**Example:**
```
iterator.reset();
WHILE(iterator.moveNext())DO
	foo := iterator.current.hashCode;
	bar := iterator.current.name;
END_WHILE
```

.. <legal notes>

legal notes
=================
| SPDX-FileCopyrightText: © 2022 ekvip automation GmbH <info@ekvip.de>
| SPDX-License-Identifier: Apache-2.0
| For details check: Apache-2.0_

.. _Apache-2.0: https://www.apache.org/licenses/LICENSE-2.0

.. </legal notes>

*)
METHOD reset
VAR CONSTANT
	NULL :__XWORD := 0;
END_VAR
THIS^.iterate(execute := FALSE);
THIS^.nextIndex := 0;
THIS^.currentObject := NULL;
END_METHOD

END_FUNCTION_BLOCK

// ---- Utils/FastSwap.TcPOU
(*
## Short summary

Fast element swap operation of two given pointers, optimized for performance.

.. <legal notes>

legal notes
=================
| SPDX-FileCopyrightText: © 2025 ekvip automation GmbH <info@ekvip.de>
| SPDX-License-Identifier: Apache-2.0
| For details check: Apache-2.0_

.. _Apache-2.0: https://www.apache.org/licenses/LICENSE-2.0

.. </legal notes>



*)

FUNCTION FastSwap
VAR_INPUT
	object1 :POINTER TO __XWORD;
	object2 :POINTER TO __XWORD;
END_VAR

RETURN(object1 = object2);
RETURN(object1 = 0 OR object2 = 0);
object1^ := object2^ XOR object1^;
object2^ := object2^ XOR object1^;
object1^ := object2^ XOR object1^;

END_FUNCTION

// ---- Lists/ArrayList/ArrayListResizingStrategy/CubicRootResizing.TcPOU
(*

## Short summary

This resizing strategy increases an capacity by a geometric factor of the cubic root of 2 (~1.26).
After three consecutive growth steps, the capacity approximately doubles, which improves the chance of reusing previously freed memory blocks and helps to reduce heap fragmentation.
The strategy is well-suited for memory-constrained or embedded environments where efficient memory reuse is more important than minimizing the number of reallocation operations.
For downsizing the capacity is reduced if the new size is less then 25 % of the current capacity. 

.. <legal notes>

legal notes
=================
| SPDX-FileCopyrightText: © 2025 ekvip automation GmbH <info@ekvip.de>
| SPDX-License-Identifier: Apache-2.0
| For details check: Apache-2.0_

.. _Apache-2.0: https://www.apache.org/licenses/LICENSE-2.0

.. </legal notes>

*)

{attribute 'enable_dynamic_creation'}
FUNCTION_BLOCK CubicRootResizing EXTENDS CNM_AbstractObject.Object IMPLEMENTS CNM_CollectionInterfaces.IResizingStrategy
VAR CONSTANT
	(* cubic root of 2 *)
	GROW_FACTOR :REAL := 1.259921049894873165;
END_VAR

(*

## Short summary

This abstract property returns the class name of the concrete object, 
which is useful for logging/debugging purpose.

.. <legal notes>

legal notes
=================
| SPDX-FileCopyrightText: © 2022 ekvip automation GmbH <info@ekvip.de>
| SPDX-License-Identifier: Apache-2.0
| For details check: Apache-2.0_

.. _Apache-2.0: https://www.apache.org/licenses/LICENSE-2.0

.. </legal notes>

*)
PROPERTY className : CNM_AbstractObject.ClassName
GET
className := 'CNM_Collections.CubicRootResizing';
END_GET
END_PROPERTY

(*

## Short summary

The method takes the requested size and the current capacity as input and determines the next suitable capacity value based on the implemented resizing strategy.
The resulting capacity is returned as newCapacity.
It returns true when a downsizing is needed within the used strategy, false if no resizing is needed.

.. <legal notes>

legal notes
=================
| SPDX-FileCopyrightText: © 2025 ekvip automation GmbH <info@ekvip.de>
| SPDX-License-Identifier: Apache-2.0
| For details check: Apache-2.0_

.. _Apache-2.0: https://www.apache.org/licenses/LICENSE-2.0

.. </legal notes>



*)
METHOD getDownscaledCapacity : BOOL
VAR_INPUT
	(* the new size that is needed *)
	requestedSize	: UDINT;
	(* the current actual size of the container *)
	currentCapacity	: UDINT;
END_VAR
VAR_OUTPUT
	(* the calculated size of the container *)
	newCapacity	: UDINT;
END_VAR
VAR CONSTANT
	SHRINKING_THRESHOLD_MULTIPLIER :UDINT := 3;
END_VAR
IF (requestedSize < THIS^.initialSize) OR_ELSE (currentCapacity = 0) THEN 
	newCapacity := THIS^.initialSize; 
ELSE 
	newCapacity := currentCapacity;  
	// gradual shrink by cubic root of 0.5 with threshold 
	WHILE ( newCapacity > SHRINKING_THRESHOLD_MULTIPLIER*requestedSize ) DO
		newCapacity := TO_UDINT(TO_REAL(newCapacity) / THIS^.GROW_FACTOR);
	END_WHILE
END_IF;

getDownscaledCapacity := (newCapacity <> currentCapacity);
END_METHOD

(*

## Short summary

The method takes the requested size and the current capacity as input and determines the next suitable capacity value based on the implemented resizing strategy.
The resulting capacity is returned as newCapacity. 
It returns true when a resizing is needed wihtin the used strategy, false if no resizing is needed.

.. <legal notes>

legal notes
=================
| SPDX-FileCopyrightText: © 2025 ekvip automation GmbH <info@ekvip.de>
| SPDX-License-Identifier: Apache-2.0
| For details check: Apache-2.0_

.. _Apache-2.0: https://www.apache.org/licenses/LICENSE-2.0

.. </legal notes>



*)
METHOD getUpscaledCapacity : BOOL
VAR_INPUT
	(* the new size that is needed *)
	requestedSize	: UDINT;
	(* the current actual size of the container *)
	currentCapacity	: UDINT;
END_VAR
VAR_OUTPUT
	(* the calculated size of the container *)
	newCapacity	: UDINT;
END_VAR
IF (requestedSize < THIS^.initialSize) THEN
	newCapacity := THIS^.initialSize;
ELSE
	newCapacity := SEL((currentCapacity = 0), newCapacity := currentCapacity, newCapacity := THIS^.initialSize);
	WHILE (newCapacity < requestedSize) DO
		newCapacity := TO_UDINT(TO_REAL(newCapacity) * THIS^.GROW_FACTOR);
	END_WHILE
END_IF
getUpscaledCapacity := (newCapacity <> currentCapacity);
END_METHOD

(*

## Short summary

This property returns an inital size for an empty new array. 

.. <legal notes>

legal notes
=================
| SPDX-FileCopyrightText: © 2025 ekvip automation GmbH <info@ekvip.de>
| SPDX-License-Identifier: Apache-2.0
| For details check: Apache-2.0_

.. _Apache-2.0: https://www.apache.org/licenses/LICENSE-2.0

.. </legal notes>



*)

PROPERTY initialSize : UDINT
GET
initialSize := 8;
END_GET
END_PROPERTY

END_FUNCTION_BLOCK

// ---- Appliers/classes/ChainedApplier.TcPOU
(*

## Short summary

An abstract class to implement the logic of Appliers for forEach. Users only need to implement apply in inherited class and should not change any other method.

.. <legal notes>

legal notes
=================
| SPDX-FileCopyrightText: © 2022 ekvip automation GmbH <info@ekvip.de>
| SPDX-License-Identifier: Apache-2.0
| For details check: Apache-2.0_

.. _Apache-2.0: https://www.apache.org/licenses/LICENSE-2.0

.. </legal notes>



*)

{attribute 'enable_dynamic_creation'}
FUNCTION_BLOCK FINAL ChainedApplier EXTENDS AbstractDisposableContainer IMPLEMENTS CNM_CollectionInterfaces.IChainedApplier
VAR
	object :CNM_AbstractObject.IObject;
END_VAR
VAR
	myactions			:ApplierList();
END_VAR

(*

## Short summary

Method to accept an object.
**Example:**
```
NumberIncrementer.accept(Number);
```

.. <legal notes>

legal notes
=================
| SPDX-FileCopyrightText: © 2022 ekvip automation GmbH <info@ekvip.de>
| SPDX-License-Identifier: Apache-2.0
| For details check: Apache-2.0_

.. _Apache-2.0: https://www.apache.org/licenses/LICENSE-2.0

.. </legal notes>



*)
METHOD accept : CNM_ReturnTypes.SingleExecutionResult
VAR_INPUT
	(*object to accept*)
	object	: CNM_AbstractObject.IObject;
END_VAR
IF(THIS^.isObjectValid(object))THEN
	THIS^.object := object;
	accept := CNM_ReturnTypes.SingleExecutionResult.SUCCESS;
ELSE
	accept := CNM_ReturnTypes.SingleExecutionResult.ERROR;	
END_IF
END_METHOD

(*

## Short summary

This property returns a list of actions/operations performed by this applier.

.. <legal notes>

legal notes
=================
| SPDX-FileCopyrightText: © 2022 ekvip automation GmbH <info@ekvip.de>
| SPDX-License-Identifier: Apache-2.0
| For details check: Apache-2.0_

.. _Apache-2.0: https://www.apache.org/licenses/LICENSE-2.0

.. </legal notes>

*)

PROPERTY actions :CNM_CollectionInterfaces.IApplierList
GET
actions := THIS^.myactions;
END_GET
END_PROPERTY

(*

## Short summary

Method to concat actions perfomed on an object. This way two (or more) Actions can be performed on data with one foreach.
All concatinated appliers can be cleared with THIS^.clear();
**Example:**
You want to double your numbers and then increment them, you would write:
```
ConcreteDoubleApplier.andThen(ConcreteIncrementApplier);
```
If you have a list with 1 2 3, after a forEach with this Applier the list will be transformed to: 3 5 7.

**Warning:**
    It is possible to create infinite loops using andThen. For example: A1.andThen(A2).andThen(A1)
	The program will go into unknown behaviour if this occurs and the foreach call may or may not work as you intended.

.. <legal notes>

legal notes
=================
| SPDX-FileCopyrightText: © 2022 ekvip automation GmbH <info@ekvip.de>
| SPDX-License-Identifier: Apache-2.0
| For details check: Apache-2.0_

.. _Apache-2.0: https://www.apache.org/licenses/LICENSE-2.0

.. </legal notes>


**Return:** ``THIS^`` `IApplier`

*)

METHOD FINAL andThen :CNM_CollectionInterfaces.IChainedApplier
VAR_INPUT
	(*the applier to be used on each object*)
	applier			:CNM_CollectionInterfaces.IApplier;
END_VAR
VAR
	chained 		:CNM_CollectionInterfaces.IChainedApplier;
	clonedActions	:CNM_CollectionInterfaces.ICollection;
	cloneObj 		:CNM_AbstractObject.IObject;
	pList 			:POINTER TO ApplierList;
END_VAR
IF(THIS^.isObjectValid(applier) AND_THEN THIS^.isObjectValid(THIS^.myactions))THEN
	IF __QUERYINTERFACE(applier, chained) THEN
		IF (chained.actions.count > 1) THEN
			IF(NOT THIS^.isEqual(applier))THEN
				__QUERYPOINTER(chained.actions, pList);
				THIS^.myactions.addAppliers(pList^.list);
			ELSE
				IF(THIS^.myactions.list.clone(clonedObject => cloneObj) = CNM_ReturnTypes.CloneResult.SUCCESS)THEN
					IF( __QUERYINTERFACE(cloneObj, clonedActions))THEN
						THIS^.myactions.addAppliers(clonedActions);					
					END_IF
					clonedActions.destruct();
				END_IF
			END_IF
		END_IF
	ELSE
		THIS^.myactions.addApplier(applier);				
	END_IF
END_IF

andThen := THIS^;
END_METHOD

(*

## Short summary

A method to apply the concrete action on the given object (THIS^.object)

.. <legal notes>

legal notes
=================
| SPDX-FileCopyrightText: © 2022 ekvip automation GmbH <info@ekvip.de>
| SPDX-License-Identifier: Apache-2.0
| For details check: Apache-2.0_

.. _Apache-2.0: https://www.apache.org/licenses/LICENSE-2.0

.. </legal notes>


**Return:** CNM_ReturnTypes.SingleExecutionState

*)

METHOD FINAL apply :CNM_ReturnTypes.SingleExecutionState
VAR_INPUT
	(*control bit to start or abort the application, should to be active until the CNM_ReturnTypes.SingleExecutionState is SUCCESS*)
	execute	:BOOL;
END_VAR
VAR_INST
	iterator 		:ForwardArrayListIterator(0);
	lastExecute 	:BOOL;
	step 			:USINT;
	returnState 	:CNM_ReturnTypes.SingleExecutionState;
	currentApplier 	:CNM_CollectionInterfaces.IApplier;
	cycleManager 	:CNM_CycleManager.SimpleCycleManager;
END_VAR
VAR
	listToAttach	:POINTER TO ArrayList;
	listReference	:REFERENCE TO ArrayList;
END_VAR
VAR CONSTANT
	INIT :DINT := CNM_ReturnTypes.DefaultSteps.STEP.INIT;
	RUN  :DINT := INIT + 1;
	GET_APPLIER :DINT := RUN + 1;
	SUCCESS :DINT := CNM_ReturnTypes.DefaultSteps.STEP.SUCCESS;
	ERROR :DINT := CNM_ReturnTypes.DefaultSteps.STEP.ERROR;
	
	STEP_IDLE :USINT := 0;
	STEP_INIT :USINT := 1;
	STEP_RUN :USINT := 2;
	STEP_DONE :USINT := 3;
	STEP_ERROR :USINT := 4;
END_VAR
cycleManager(execute := execute);

CASE cycleManager.step.current OF
INIT:
	cycleManager.configuration.sequence.requireSuccessStep := FALSE;
	__QUERYPOINTER(THIS^.myactions.list, listToAttach);
	listReference REF= listToAttach^;
	iterator.attachArrayList(listReference);
	iterator.reset();
	IF(iterator.moveNext() AND_THEN __QUERYINTERFACE(iterator.current, currentApplier))THEN
		currentApplier.accept(THIS^.object);
		currentApplier.apply(FALSE);
		currentApplier.apply(TRUE);
		cycleManager.proceed();
	ELSE
		cycleManager.proceedWith(SUCCESS);
	END_IF
	
RUN:
	CASE currentApplier.apply(TRUE) OF
	CNM_ReturnTypes.SingleExecutionState.SUCCESS:	
		cycleManager.proceed();
	CNM_ReturnTypes.SingleExecutionState.ABORTED,
	CNM_ReturnTypes.SingleExecutionState.ERROR:
		cycleManager.proceedWith(ERROR);
	ELSE
		;// do nothing, stay in RUN
	END_CASE
	
GET_APPLIER:
	IF(iterator.moveNext() AND_THEN __QUERYINTERFACE(iterator.current, currentApplier))THEN
		currentApplier.accept(THIS^.object);
		currentApplier.apply(FALSE);
		currentApplier.apply(TRUE);
		cycleManager.proceedWith(RUN);
	ELSE
		cycleManager.proceedWith(SUCCESS);
	END_IF
	
END_CASE

apply := cycleManager.state;
END_METHOD

(*

## Short summary

This abstract property returns the class name of the concrete object, 
which is useful to check the class name for ``__DELETE``.

.. <legal notes>

legal notes
=================
| SPDX-FileCopyrightText: © 2022 ekvip automation GmbH <info@ekvip.de>
| SPDX-License-Identifier: Apache-2.0
| For details check: Apache-2.0_

.. _Apache-2.0: https://www.apache.org/licenses/LICENSE-2.0

.. </legal notes>

*)

PROPERTY className :CNM_AbstractObject.ClassName
GET
className := 'ChainedApplier';
END_GET
END_PROPERTY

(*

## Short summary

This method is called in the destruct method and is intended to zero all references and interfaces that should not be destructed. 
To delete the collection with all its contents, use deepDestruct() instead of destruct().

.. <legal notes>

legal notes
=================
| SPDX-FileCopyrightText: © 2025 ekvip automation GmbH <info@ekvip.de>
| SPDX-License-Identifier: Apache-2.0
| For details check: Apache-2.0_

.. _Apache-2.0: https://www.apache.org/licenses/LICENSE-2.0

.. </legal notes>

*)
METHOD PROTECTED clearContents
VAR CONSTANT
	NULL	: __XWORD := 0;
END_VAR
THIS^.object := NULL;
END_METHOD

(*

## Short summary

Mark the object as deleted, as it staiys in the memory.

.. <legal notes>

legal notes
=================
| SPDX-FileCopyrightText: © 2022 ekvip automation GmbH <info@ekvip.de>
| SPDX-License-Identifier: Apache-2.0
| For details check: Apache-2.0_

.. _Apache-2.0: https://www.apache.org/licenses/LICENSE-2.0

.. </legal notes>

*)
METHOD FB_Exit : BOOL
VAR_INPUT
	(* TRUE: the exit method is called in order to leave the instance which will be copied afterwards (online change).*)
	bInCopyCode	: BOOL;
END_VAR
IF THIS^.isObjectValid(THIS^.object) THEN
	THIS^.object.deepDestruct();
END_IF
END_METHOD

(*

## Short summary

The constructor ``FB_init`` is needed to create an unique hash code.
The hash code is a pseudo random number create with a [xorshift](https://en.wikipedia.org/wiki/Xorshift) algorithm.
It can be overwritten on derivations, because it will be called implicit, ``SUPER^.FB_init()`` is not required.
For more information check: [Behavoir with derived function blocks](https://infosys.beckhoff.com/content/1033/tc3_plc_intro/5482088715.html?id=6983869892358031022).

.. <legal notes>

legal notes
=================
| SPDX-FileCopyrightText: © 2022 ekvip automation GmbH <info@ekvip.de>
| SPDX-License-Identifier: Apache-2.0
| For details check: Apache-2.0_

.. _Apache-2.0: https://www.apache.org/licenses/LICENSE-2.0

.. </legal notes>



*)
METHOD FB_init : BOOL
VAR_INPUT
	(* if TRUE, the retain variables are initialized (warm start / cold start)*)
	bInitRetains	: BOOL;
	(* if TRUE, the instance afterwards gets moved into the copy code (online change) *)
	bInCopyCode	: BOOL;
	firstApplier :CNM_CollectionInterfaces.IApplier;
	secondApplier :CNM_CollectionInterfaces.IApplier;
END_VAR
THIS^.myactions.clear();
THIS^.myactions.addApplier(firstApplier);
THIS^.myactions.addApplier(secondApplier);
END_METHOD

END_FUNCTION_BLOCK

// ---- BinaryTree/BBSTIterator/classes/BfsBbstIterator.TcPOU
(*

## Short summary

This class implements the breadth first iteration strategy for balanced binary search trees.

.. <legal notes>

legal notes
=================
| SPDX-FileCopyrightText: © 2024 ekvip automation GmbH <info@ekvip.de>
| SPDX-License-Identifier: Apache-2.0
| For details check: Apache-2.0_

.. _Apache-2.0: https://www.apache.org/licenses/LICENSE-2.0

.. </legal notes>

*)

{attribute 'enable_dynamic_creation'}
FUNCTION_BLOCK BfsBbstIterator EXTENDS AbstractBalancedBinarySearchTreeIterator

PROPERTY className :CNM_AbstractObject.ClassName
GET
className := 'CNM_Collections.BFS_BBSTIterator';
END_GET
END_PROPERTY

(*

## Short summary

Gets the next Node that iterate should process.

.. <legal notes>

legal notes
=================
| SPDX-FileCopyrightText: © 2022 ekvip automation GmbH <info@ekvip.de>
| SPDX-License-Identifier: Apache-2.0
| For details check: Apache-2.0_

.. _Apache-2.0: https://www.apache.org/licenses/LICENSE-2.0

.. </legal notes>


**Return:** ``TRUE`` a valid node existed, ``FALSE`` no node for iteration existed

*)

METHOD PROTECTED getNextTreeNode : BOOL
VAR_OUTPUT
	node	:CNM_CollectionInterfaces.IBinaryTreeNode;
END_VAR
VAR
	tmpObject :CNM_AbstractObject.IObject;
END_VAR
tmpObject := THIS^.nodeList.dequeue();
__QUERYINTERFACE(tmpObject, node);
getNextTreeNode := THIS^.isObjectValid(node);
END_METHOD

(*

## Short summary

This method appends (if they exists) the left and right child of the node to the nodelist.

.. <legal notes>

legal notes
=================
| SPDX-FileCopyrightText: © 2022 ekvip automation GmbH <info@ekvip.de>
| SPDX-License-Identifier: Apache-2.0
| For details check: Apache-2.0_

.. _Apache-2.0: https://www.apache.org/licenses/LICENSE-2.0

.. </legal notes>



*)

METHOD PROTECTED processNode
VAR_INPUT
	nodeToProcess	: CNM_CollectionInterfaces.IBinaryTreeNode;
END_VAR
IF(nodeToProcess.leftChild <> 0)THEN
	THIS^.nodeList.append(nodeToProcess.leftChild);
END_IF
IF(nodeToProcess.rightChild <> 0)THEN
	THIS^.nodeList.append(nodeToProcess.rightChild);
END_IF
END_METHOD

END_FUNCTION_BLOCK

// ---- BinaryTree/BBSTIterator/classes/DfsBbstIterator.TcPOU
(*

## Short summary

This class implements the depth first iteration strategy for balanced binary search trees.

.. <legal notes>

legal notes
=================
| SPDX-FileCopyrightText: © 2024 ekvip automation GmbH <info@ekvip.de>
| SPDX-License-Identifier: Apache-2.0
| For details check: Apache-2.0_

.. _Apache-2.0: https://www.apache.org/licenses/LICENSE-2.0

.. </legal notes>

*)


{attribute 'enable_dynamic_creation'}
FUNCTION_BLOCK DfsBbstIterator EXTENDS AbstractBalancedBinarySearchTreeIterator

PROPERTY className : CNM_AbstractObject.ClassName
GET
className := 'CNM_Collections.DFS_BBSTIterator';
END_GET
END_PROPERTY

(*

## Short summary

Gets the next Node that iterate should process.

.. <legal notes>

legal notes
=================
| SPDX-FileCopyrightText: © 2022 ekvip automation GmbH <info@ekvip.de>
| SPDX-License-Identifier: Apache-2.0
| For details check: Apache-2.0_

.. _Apache-2.0: https://www.apache.org/licenses/LICENSE-2.0

.. </legal notes>


**Return:** ``TRUE`` a valid node existed, ``FALSE`` no node for iteration existed

*)

METHOD PROTECTED getNextTreeNode : BOOL
VAR_OUTPUT
	node	: CNM_CollectionInterfaces.IBinaryTreeNode;
END_VAR
VAR
	tmpObject :CNM_AbstractObject.IObject;
END_VAR
tmpObject := THIS^.nodeList.pop();
__QUERYINTERFACE(tmpObject, node);
getNextTreeNode := THIS^.isObjectValid(node);
END_METHOD

(*

## Short summary

This method appends (if they exists) the left and right child of the node to the nodelist.

.. <legal notes>

legal notes
=================
| SPDX-FileCopyrightText: © 2022 ekvip automation GmbH <info@ekvip.de>
| SPDX-License-Identifier: Apache-2.0
| For details check: Apache-2.0_

.. _Apache-2.0: https://www.apache.org/licenses/LICENSE-2.0

.. </legal notes>



*)

METHOD PROTECTED processNode
VAR_INPUT
	nodeToProcess	: CNM_CollectionInterfaces.IBinaryTreeNode;
END_VAR
IF(nodeToProcess.rightChild <> 0)THEN
	THIS^.nodeList.append(nodeToProcess.rightChild);
END_IF
IF(nodeToProcess.leftChild <> 0)THEN
	THIS^.nodeList.append(nodeToProcess.leftChild);
END_IF
END_METHOD

END_FUNCTION_BLOCK

// ---- Lists/ArrayList/ArrayListIterator/classes/InverseArrayListIterator.TcPOU
(*

## Short summary

This class can be used as a simple inverse iterator for array lists. It iterates from last element to first element.

.. <legal notes>

legal notes
=================
| SPDX-FileCopyrightText: © 2024 ekvip automation GmbH <info@ekvip.de>
| SPDX-License-Identifier: Apache-2.0
| For details check: Apache-2.0_

.. _Apache-2.0: https://www.apache.org/licenses/LICENSE-2.0

.. </legal notes>



*)

{attribute 'enable_dynamic_creation'}
FUNCTION_BLOCK InverseArrayListIterator EXTENDS AbstractArrayListIterator

PROPERTY className :CNM_AbstractObject.ClassName
GET
className := 'InverseArrayListIterator';
END_GET
END_PROPERTY

(*

## Short summary

The constructor ``FB_init`` is needed to create an unique hash code.
The hash code is a pseudo random number create with a [xorshift](https://en.wikipedia.org/wiki/Xorshift) algorithm.
It can be overwritten on derivations, because it will be called implicit, ``SUPER^.FB_init()`` is not required.
For more information check: [Behavoir with derived function blocks](https://infosys.beckhoff.com/content/1033/tc3_plc_intro/5482088715.html?id=6983869892358031022).

.. <legal notes>

legal notes
=================
| SPDX-FileCopyrightText: © 2022 ekvip automation GmbH <info@ekvip.de>
| SPDX-License-Identifier: Apache-2.0
| For details check: Apache-2.0_

.. _Apache-2.0: https://www.apache.org/licenses/LICENSE-2.0

.. </legal notes>



*)
METHOD FB_init : BOOL
VAR_INPUT
	(* if TRUE, the retain variables are initialized (warm start / cold start)*)
	bInitRetains	: BOOL;
	(* if TRUE, the instance afterwards gets moved into the copy code (online change) *)
	bInCopyCode	: BOOL;
	(* the array list which should be iterated, can be 0 *)
	arrayList :REFERENCE TO ArrayList;
END_VAR
THIS^.direction := IterationDirection.BACKWARD;
END_METHOD

END_FUNCTION_BLOCK

// ---- Lists/ArrayList/ArrayListResizingStrategy/CubicRootUpsizeOnly.TcPOU
(*

## Short summary

This resizing strategy increases an capacity by a geometric factor of the cubic root of 2 (~1.26).
After three consecutive growth steps, the capacity approximately doubles, which improves the chance of reusing previously freed memory blocks and helps to reduce heap fragmentation.
The strategy is well-suited for memory-constrained or embedded environments where efficient memory reuse is more important than minimizing the number of reallocation operations.
This strategy will not downsize the capacity, this means there is no shrinking possible. 
It can be used for starage with constant max size, e.g. warehouse applications or shelfs.

.. <legal notes>

legal notes
=================
| SPDX-FileCopyrightText: © 2025 ekvip automation GmbH <info@ekvip.de>
| SPDX-License-Identifier: Apache-2.0
| For details check: Apache-2.0_

.. _Apache-2.0: https://www.apache.org/licenses/LICENSE-2.0

.. </legal notes>

*)

{attribute 'enable_dynamic_creation'}
FUNCTION_BLOCK CubicRootUpsizeOnly EXTENDS CNM_AbstractObject.Object IMPLEMENTS CNM_CollectionInterfaces.IResizingStrategy
VAR CONSTANT
	(* cubic root of 2 *)
	GROW_FACTOR :REAL := 1.259921049894873165;
END_VAR

(*

## Short summary

This abstract property returns the class name of the concrete object, 
which is useful for logging/debugging purpose.

.. <legal notes>

legal notes
=================
| SPDX-FileCopyrightText: © 2022 ekvip automation GmbH <info@ekvip.de>
| SPDX-License-Identifier: Apache-2.0
| For details check: Apache-2.0_

.. _Apache-2.0: https://www.apache.org/licenses/LICENSE-2.0

.. </legal notes>

*)
PROPERTY className : CNM_AbstractObject.ClassName
GET
className := 'CNM_Collections.CubicRootUpsizeOnly';
END_GET
END_PROPERTY

(*

## Short summary

The method takes the requested size and the current capacity as input and determines the next suitable capacity value based on the implemented resizing strategy.
The resulting capacity is returned as newCapacity.
It returns true when a downsizing is needed within the used strategy, false if no resizing is needed.

.. <legal notes>

legal notes
=================
| SPDX-FileCopyrightText: © 2025 ekvip automation GmbH <info@ekvip.de>
| SPDX-License-Identifier: Apache-2.0
| For details check: Apache-2.0_

.. _Apache-2.0: https://www.apache.org/licenses/LICENSE-2.0

.. </legal notes>



*)
METHOD getDownscaledCapacity : BOOL
VAR_INPUT
	(* the new size that is needed *)
	requestedSize	: UDINT;
	(* the current actual size of the container *)
	currentCapacity	: UDINT;
END_VAR
VAR_OUTPUT
	(* the calculated size of the container *)
	newCapacity	: UDINT;
END_VAR
newCapacity := currentCapacity;
getDownscaledCapacity := FALSE;
END_METHOD

(*

## Short summary

The method takes the requested size and the current capacity as input and determines the next suitable capacity value based on the implemented resizing strategy.
The resulting capacity is returned as newCapacity. 
It returns true when a resizing is needed wihtin the used strategy, false if no resizing is needed.

.. <legal notes>

legal notes
=================
| SPDX-FileCopyrightText: © 2025 ekvip automation GmbH <info@ekvip.de>
| SPDX-License-Identifier: Apache-2.0
| For details check: Apache-2.0_

.. _Apache-2.0: https://www.apache.org/licenses/LICENSE-2.0

.. </legal notes>



*)
METHOD getUpscaledCapacity : BOOL
VAR_INPUT
	(* the new size that is needed *)
	requestedSize	: UDINT;
	(* the current actual size of the container *)
	currentCapacity	: UDINT;
END_VAR
VAR_OUTPUT
	(* the calculated size of the container *)
	newCapacity	: UDINT;
END_VAR
IF (requestedSize < THIS^.initialSize) THEN
	newCapacity := THIS^.initialSize;
ELSE
	newCapacity := SEL((currentCapacity = 0), newCapacity := currentCapacity, newCapacity := THIS^.initialSize);
	WHILE (newCapacity < requestedSize) DO
		newCapacity := TO_UDINT(TO_REAL(newCapacity) * THIS^.GROW_FACTOR);
	END_WHILE
END_IF
getUpscaledCapacity := (newCapacity <> currentCapacity);
END_METHOD

(*

## Short summary

This property returns an inital size for an empty new array. 

.. <legal notes>

legal notes
=================
| SPDX-FileCopyrightText: © 2025 ekvip automation GmbH <info@ekvip.de>
| SPDX-License-Identifier: Apache-2.0
| For details check: Apache-2.0_

.. _Apache-2.0: https://www.apache.org/licenses/LICENSE-2.0

.. </legal notes>



*)

PROPERTY initialSize : UDINT
GET
initialSize := 8;
END_GET
END_PROPERTY

END_FUNCTION_BLOCK

// ---- Lists/ArrayList/ArrayListSorter/ArrayListTwinSorter.TcPOU
(*

## Short summary

Implementation of TwinSort algorithm for ArrayList with performance optimizations.
TwinSort is an adaptive, stable mergesort variant that optimizes naturally ordered pairs
and reverse-ordered sequences through intelligent preprocessing.

Key features:
- Preprocessing phase creates naturally sorted pairs
- Reverses descending sequences to exploit existing order
- Adaptive merge strategy with optimized boundary detection
- O(n log n) worst case, O(n) best case for sorted data
- Stable sort (maintains relative order of equal elements)
- Optimized for real-world data patterns

Performance optimizations in this version:
- Pre-allocated merge buffer to avoid repeated allocations
- Buffer size tracking with 25% extra space to minimize reallocations
- WHILE loops instead of FOR loops for better performance
- State preservation between cycles to avoid redundant work
- Optimized buffer management with size-based pre-allocation

The algorithm works by:
1. Preprocessing: Identify and sort adjacent pairs, reverse descending sequences
2. Adaptive merging: Skip unnecessary merges when sequences are already ordered
3. Boundary optimization: Reduce work by detecting optimal merge boundaries
4. Memory-efficient: Pre-allocated buffer with intelligent sizing

Based on research from lost-and-found-in-arrays repository, adapted for
CNM Collections framework with real-time constraints and performance optimizations.

.. <legal notes>

legal notes
=================
| SPDX-FileCopyrightText: © 2025 ekvip automation GmbH <info@ekvip.de>
| SPDX-License-Identifier: Apache-2.0
| For details check: Apache-2.0_

.. _Apache-2.0: https://www.apache.org/licenses/LICENSE-2.0

.. </legal notes>



*)

{attribute 'enable_dynamic_creation'}
FUNCTION_BLOCK FINAL ArrayListTwinSorter EXTENDS AbstractArrayListSorter
VAR
	// Merge buffer for temporary storage during merges - pre-allocated
	mergeBuffer :POINTER TO CNM_AbstractObject.IObject;
END_VAR

(*

## Short summary

This abstract property returns the class name of the concrete object, 
which is useful to check the class name for ``__DELETE``.

.. <legal notes>

legal notes
=================
| SPDX-FileCopyrightText: © 2022 ekvip automation GmbH <info@ekvip.de>
| SPDX-License-Identifier: Apache-2.0
| For details check: Apache-2.0_

.. _Apache-2.0: https://www.apache.org/licenses/LICENSE-2.0

.. </legal notes>

*)
PROPERTY className : CNM_AbstractObject.ClassName
GET
className := 'CNM_Collections.ArrayListTwinSorter';
END_GET
END_PROPERTY

(*

## Short summary

This method is called in the destruct method and is intended to zero all references and interfaces that should not be destructed. 
To delete the collection with all its contents, use deepDestruct() instead of destruct().

.. <legal notes>

legal notes
=================
| SPDX-FileCopyrightText: © 2025 ekvip automation GmbH <info@ekvip.de>
| SPDX-License-Identifier: Apache-2.0
| For details check: Apache-2.0_

.. _Apache-2.0: https://www.apache.org/licenses/LICENSE-2.0

.. </legal notes>

*)
METHOD PROTECTED clearContents
END_METHOD

(*

## Short summary

This method is used to create a new instance
of the object which has the same internal state as the object.

.. <legal notes>

legal notes
=================
| SPDX-FileCopyrightText: © 2022 ekvip automation GmbH <info@ekvip.de>
| SPDX-License-Identifier: Apache-2.0
| For details check: Apache-2.0_

.. _Apache-2.0: https://www.apache.org/licenses/LICENSE-2.0

.. </legal notes>


**Return:**``CNM_ReturnTypes.CloneResult.SUCCESS``: new object clone was created,
``CNM_ReturnTypes.CloneResult.FAILED``: object clone failed

*)
METHOD clone : CNM_AbstractObject.CNM_ReturnTypes.CloneResult
VAR
	newSorter :POINTER TO ArrayListTwinSorter;
END_VAR
VAR_OUTPUT
	(* new object instance or NULL if somthing went wrong *)
	clonedObject	: CNM_AbstractObject.IObject;
END_VAR
newSorter := __NEW(ArrayListTwinSorter());

IF (newSorter = 0) THEN
	clone := CNM_ReturnTypes.CloneResult.FAILED;
	clonedObject := 0;
ELSE
	clone := CNM_ReturnTypes.CloneResult.SUCCESS;
	clonedObject := newSorter^;
	THIS^.prepareClonedSorter(newSorter^);
END_IF
END_METHOD

(*

## Short summary

Mark the object as deleted, as it staiys in the memory.

.. <legal notes>

legal notes
=================
| SPDX-FileCopyrightText: © 2022 ekvip automation GmbH <info@ekvip.de>
| SPDX-License-Identifier: Apache-2.0
| For details check: Apache-2.0_

.. _Apache-2.0: https://www.apache.org/licenses/LICENSE-2.0

.. </legal notes>

*)
METHOD FB_Exit : BOOL
VAR_INPUT
	(* TRUE: the exit method is called in order to leave the instance which will be copied afterwards (online change).*)
	bInCopyCode	: BOOL;
END_VAR
__DELETE(THIS^.mergeBuffer);
END_METHOD

(*

## Short summary

This method sorts the data structure instantly within one call. 
It uses the passed Comparator to sort the structure or the compareTo of the contained Objects if no comparator is passed.

.. <legal notes>

legal notes
=================
| SPDX-FileCopyrightText: © 2025 ekvip automation GmbH <info@ekvip.de>
| SPDX-License-Identifier: Apache-2.0
| For details check: Apache-2.0_

.. _Apache-2.0: https://www.apache.org/licenses/LICENSE-2.0

.. </legal notes>


**Return:**``ERROR``: Sort was not able to finish 
	``SUCCESS``: Sorting was finished succesfully

*)
METHOD instantSort : CNM_CollectionInterfaces.CNM_ReturnTypes.SingleExecutionResult
VAR_INPUT
	(*The size of the list to be sorted*)
	size	: UDINT;
	(*the container, that contains the list elements*)
	container	: POINTER TO CNM_CollectionInterfaces.CNM_AbstractObject.IObject;
	(*the comparator that should be used for the sort. Must not be changed while sort is in process*)
	comparator	: CNM_CollectionInterfaces.CNM_AbstractObject.IComparator := 0;
END_VAR
VAR_IN_OUT
	(*the current version of the list, must change when the data in the list changes *)
	currentListVersion	: __XWORD;
END_VAR
VAR
	mergeWidth :UDINT := 2;
	preprocessResult :CNM_ReturnTypes.SingleExecutionResult; 
END_VAR
mergeWidth := 2;
instantSort := CNM_ReturnTypes.SingleExecutionResult.SUCCESS;
RETURN(size <= 1);
THIS^.setComparator(comparator);
preprocessResult := THIS^.preprocessElements(container, size);
currentListVersion := currentListVersion + 1;
CASE preprocessResult OF 
CNM_ReturnTypes.SingleExecutionResult.SUCCESS:
	IF THIS^.mergeBuffer <> 0 THEN
		__DELETE(THIS^.mergeBuffer);
	END_IF
	THIS^.mergeBuffer := __NEW(__XWORD, SHR(size + 1, 1));
CNM_ReturnTypes.SingleExecutionResult.ABORTED:
	__DELETE(THIS^.mergeBuffer);
	instantSort := CNM_ReturnTypes.SingleExecutionResult.SUCCESS;
	RETURN;
ELSE
	__DELETE(THIS^.mergeBuffer);
	instantSort := CNM_ReturnTypes.SingleExecutionResult.ERROR;
	RETURN;
END_CASE

WHILE mergeWidth < size DO 
	THIS^.merge( container, size, mergeWidth);
	mergeWidth := SHL(mergeWidth, 1);
END_WHILE
__DELETE(THIS^.mergeBuffer);
	
instantSort := CNM_ReturnTypes.SingleExecutionResult.SUCCESS;
END_METHOD


(*

## Short summary

Inverts the order of the elements inside the list. 
Does not apply any kind of sorting, only reverses the elements in the list.

.. <legal notes>

legal notes
=================
| SPDX-FileCopyrightText: © 2022 ekvip automation GmbH <info@ekvip.de>
| SPDX-License-Identifier: Apache-2.0
| For details check: Apache-2.0_

.. _Apache-2.0: https://www.apache.org/licenses/LICENSE-2.0

.. </legal notes>

*)

METHOD invertArray
VAR_INPUT
	addressFirstElement	:POINTER TO __XWORD;
	addressLastElement	:POINTER TO __XWORD;
END_VAR
VAR
	midLower	:POINTER TO __XWORD;
	midUpper	:POINTER TO __XWORD;
	loop		:__XWORD;
	size 		:UDINT;
END_VAR
VAR CONSTANT
	REGISTER_SIZE :__XWORD := SIZEOF(__XWORD);
END_VAR
CASE (size := SHR((addressLastElement - addressFirstElement), log2(REGISTER_SIZE)) + 1) OF
0,1: RETURN;
2,3: fastSwap(addressFirstElement, addressLastElement);RETURN;
END_CASE


loop := SHR(addressLastElement - addressFirstElement, SHR(REGISTER_SIZE,2) + 2);

midLower := addressFirstElement + (loop * REGISTER_SIZE);
midUpper := addressLastElement - (loop * REGISTER_SIZE);

IF ((loop AND 1) <> 0) THEN
	midLower^ := midLower^ XOR midUpper^;
	midUpper^ := midLower^ XOR midUpper^;
	midLower^ := midLower^ XOR midUpper^;
	midLower := midLower - REGISTER_SIZE;
	midUpper := midUpper + REGISTER_SIZE;
	loop := loop - 1;
END_IF;

loop := MAX(SHR(loop, 1), 1);
	
REPEAT
	addressFirstElement^ := addressFirstElement^ XOR addressLastElement^;
	addressLastElement^ := addressFirstElement^ XOR addressLastElement^;
	addressFirstElement^ := addressFirstElement^ XOR addressLastElement^;
	midLower^ := midLower^ XOR midUpper^;
	midUpper^ := midLower^ XOR midUpper^;
	midLower^ := midLower^ XOR midUpper^;
	midLower := midLower - REGISTER_SIZE;
	midUpper := midUpper + REGISTER_SIZE;
	addressFirstElement := addressFirstElement + REGISTER_SIZE;
	addressLastElement := addressLastElement - REGISTER_SIZE;
	loop := loop - 1;
UNTIL (loop = 0) END_REPEAT
END_METHOD

(*

## Short summary

Merges two adjacent sorted sequences with adaptive boundary optimization.
Uses cycle-limited execution for real-time constraints.

.. <legal notes>

legal notes
=================
| SPDX-FileCopyrightText: © 2025 ekvip automation GmbH <info@ekvip.de>
| SPDX-License-Identifier: Apache-2.0
| For details check: Apache-2.0_

.. _Apache-2.0: https://www.apache.org/licenses/LICENSE-2.0

.. </legal notes>


**Return:** TRUE if merge completed, FALSE if needs more cycles

*)

METHOD PRIVATE merge : BOOL
VAR_INPUT
	container :POINTER TO CNM_AbstractObject.IObject;
	arraySize :UDINT;
	mergeWidth :UDINT;
END_VAR
VAR
	leftEnd, leftStart, rightStart, rightEnd :LINT;
	bufferEnd, bufferIndex :LINT;
	copyCount :__XWORD;
	i :__XWORD;
	offset :LINT;
	bufferWriteStart :LINT := 0;
	rightIndex :LINT;
END_VAR
offset := 0;
WHILE ((offset + mergeWidth) < arraySize) DO
	leftStart := offset;
	leftEnd := leftStart + mergeWidth - 1;
	IF (THIS^.compareElements(container[leftEnd], container[leftEnd + 1]) <= CNM_ReturnTypes.ComparationResult.EQUAL) THEN
		offset := offset + SHL(mergeWidth,1);
		CONTINUE;
	END_IF
	IF ((offset + SHL(mergeWidth,1)) <= arraySize) THEN
		bufferEnd := bufferWriteStart + mergeWidth;
		rightEnd := (leftStart + SHL(mergeWidth,1));
	ELSE
		bufferEnd := (bufferWriteStart + arraySize - (offset + mergeWidth));
		rightEnd := arraySize;
	END_IF
	rightIndex := rightEnd - 1;
	WHILE (THIS^.compareElements(container[leftEnd], container[rightIndex]) <= CNM_ReturnTypes.ComparationResult.EQUAL) DO
		rightEnd := rightEnd - 1;
		bufferEnd := bufferEnd - 1;
		rightIndex := rightIndex - 1;
	END_WHILE
	bufferIndex := bufferWriteStart;
	rightIndex := leftStart + mergeWidth;
	WHILE (bufferIndex < bufferEnd) DO
		THIS^.mergeBuffer[bufferIndex] := container[rightIndex];
		bufferIndex := bufferIndex + 1;
		rightIndex := rightIndex + 1;
	END_WHILE
	bufferIndex := bufferIndex - 1;
	rightIndex := leftStart + mergeWidth - 1;
	leftEnd := rightEnd - 1;
	IF (THIS^.compareElements(container[leftStart], container[leftStart + mergeWidth]) <= CNM_ReturnTypes.ComparationResult.EQUAL) THEN
		container[leftEnd] := container[rightIndex];
		leftEnd := leftEnd - 1;
		rightIndex := rightIndex - 1;
		WHILE (bufferIndex >= bufferWriteStart) DO
			WHILE (THIS^.compareElements(container[rightIndex], THIS^.mergeBuffer[bufferIndex]) = CNM_ReturnTypes.ComparationResult.GREATER) DO
				container[leftEnd] := container[rightIndex];
				leftEnd := leftEnd - 1;
				rightIndex := rightIndex - 1;
			END_WHILE
			container[leftEnd] := THIS^.mergeBuffer[bufferIndex];
			leftEnd := leftEnd - 1;
			bufferIndex := bufferIndex - 1;
		END_WHILE
	ELSE
		container[leftEnd] := container[rightIndex];
		leftEnd := leftEnd - 1;
		rightIndex := rightIndex - 1;
		WHILE (rightIndex >= leftStart) DO
			WHILE (THIS^.compareElements(container[rightIndex], THIS^.mergeBuffer[bufferIndex]) <= CNM_ReturnTypes.ComparationResult.EQUAL) DO
				container[leftEnd] := THIS^.mergeBuffer[bufferIndex];
				leftEnd := leftEnd - 1;
				bufferIndex := bufferIndex - 1;
			END_WHILE
			container[leftEnd] := container[rightIndex];
			leftEnd := leftEnd - 1;
			rightIndex := rightIndex - 1;
		END_WHILE
		WHILE (bufferIndex >= bufferWriteStart) DO
			container[leftEnd] := THIS^.mergeBuffer[bufferIndex];
			leftEnd := leftEnd - 1;
			bufferIndex := bufferIndex - 1;
		END_WHILE
	END_IF
	offset := offset + SHL(mergeWidth,1);
END_WHILE
END_METHOD

(*

## Short summary

Preprocessing phase that creates naturally sorted pairs and reverses
descending sequences to optimize the merge phase.

.. <legal notes>

legal notes
=================
| SPDX-FileCopyrightText: © 2025 ekvip automation GmbH <info@ekvip.de>
| SPDX-License-Identifier: Apache-2.0
| For details check: Apache-2.0_

.. _Apache-2.0: https://www.apache.org/licenses/LICENSE-2.0

.. </legal notes>


**Return:** ``SUCCESS``: list ready for sorting 
		``ERROR``: invalid container reference 
		``ABORTED``: list is already sorted

*)

METHOD PRIVATE preprocessElements :CNM_ReturnTypes.SingleExecutionResult
VAR_INPUT
	container :POINTER TO CNM_AbstractObject.IObject;
	numberOfElements :UDINT;
END_VAR
VAR
	index :UDINT := 0;
	swapCount :__XWORD;
	i :__XWORD;
	upper :POINTER TO __XWORD;
	lower :POINTER TO __XWORD;
	end, start :__XINT;
END_VAR
VAR CONSTANT
	POINTER_SIZE_IN_BYTE :__XWORD := SIZEOF(__XWORD);
END_VAR
preprocessElements := CNM_ReturnTypes.SingleExecutionResult.ERROR;
RETURN(container = 0);
end := numberOfElements - 2;
WHILE (index <= end) DO
	IF (THIS^.compareElements(container[index], container[index+1]) <= CNM_ReturnTypes.ComparationResult.EQUAL) THEN
		index := index + 2;
		CONTINUE;
	END_IF
	start := index;
	index := index + 2;
	WHILE (TRUE) DO
		IF (index > end) THEN
			IF (start = 0) THEN
				IF (
					((numberOfElements AND 1) = 0)
					OR_ELSE  (THIS^.compareElements(container[index-1], container[index]) = CNM_ReturnTypes.ComparationResult.GREATER)
				) THEN
					end := numberOfElements - 1; 
					THIS^.invertArray(ADR(container[start]), ADR(container[end]));
					preprocessElements := CNM_ReturnTypes.SingleExecutionResult.ABORTED;
					RETURN;
				END_IF
			END_IF
			EXIT;
		END_IF
		IF (THIS^.compareElements(container[index], container[index+1]) = CNM_ReturnTypes.ComparationResult.GREATER) THEN
			IF 	(THIS^.compareElements(container[index-1], container[index]) = CNM_ReturnTypes.ComparationResult.GREATER) THEN
				index := index + 2;
				CONTINUE;
			END_IF
			FastSwap(ADR(container[index]), ADR(container[index + 1]));
		END_IF
		EXIT;
	END_WHILE
	end := index - 1;
	WHILE (start < end) DO
		FastSwap(ADR(container[start]), ADR(container[end]));
		start := start + 1;
		end := end - 1;
	END_WHILE
	end := numberOfElements - 2;
	index := index + 2;
END_WHILE;
preprocessElements := CNM_ReturnTypes.SingleExecutionResult.SUCCESS;
END_METHOD

(*

## Short summary

This method sorts the ArrayList using the TwinSort algorithm.
It uses the passed Comparator to sort the structure.
This can take many cycles and should be called until the ExecutionState is no longer ``BUSY``.

.. <legal notes>

legal notes
=================
| SPDX-FileCopyrightText: © 2025 ekvip automation GmbH <info@ekvip.de>
| SPDX-License-Identifier: Apache-2.0
| For details check: Apache-2.0_

.. _Apache-2.0: https://www.apache.org/licenses/LICENSE-2.0

.. </legal notes>


**Return:** ``ABORTED``: While sort was pending, execute had a falling edge,
	``BUSY``: Sort is in progress
	``ERROR``: Sort was not able to finish (e.g. List changed)
	``IDLE``: Currently no sort in progress
	``SUCCESS``: Sorting was finished 

*)
METHOD sort : CNM_ReturnTypes.SingleExecutionState
VAR_INPUT
	(*control bit to start or abort the sorting, needs to be active until the ExecutionState is SUCCESS*)
	execute		:BOOL;
	(*The size of the list to be sorted*)
	size 		:UDINT;
	(*the container, that contains the list elements*)
	container	:POINTER TO CNM_AbstractObject.IObject;
	(*the comparator that should be used for the sort. Must not be changed while sort is in process*)
	comparator :CNM_AbstractObject.IComparator := 0;
END_VAR
VAR_IN_OUT
	(*the current version of the list, must change when the data in the list changes *)
	currentListVersion :__XWORD;
END_VAR
VAR_INST
	lastListChangeIndex :__XWORD;
	// Merge state
	cycleManager	:CNM_CycleManager.SimpleCycleManager;
	mergeWidth 		:UDINT;
END_VAR
VAR
	preprocessResult :CNM_ReturnTypes.SingleExecutionResult;
END_VAR
VAR CONSTANT
	INIT :DINT := CNM_ReturnTypes.DefaultSteps.STEP.INIT;
	PRE_PROCESSING :DINT := INIT + 1;
	MERGING :DINT := PRE_PROCESSING + 1;
	SUCCESS :DINT := CNM_ReturnTypes.DefaultSteps.STEP.SUCCESS;
	ERROR :DINT := CNM_ReturnTypes.DefaultSteps.STEP.ERROR;
END_VAR
cycleManager.update(execute := execute);
IF cycleManager.step.current > INIT THEN
	cycleManager.assert.bitNumber.x.valueIsEqualTo(
		currentValue := currentListVersion, 
		expectedValue := lastListChangeIndex, 
		message := 'list has changed during pending sorting'
	);
END_IF

CASE cycleManager.step.current OF 
INIT:
	cycleManager.configuration.sequence.requireSuccessStep := FALSE;
	THIS^.setComparator(comparator);
	lastListChangeIndex := currentListVersion;
	// Initialize state
	mergeWidth := 2;
	cycleManager.proceedWith(SEL((size <= 1), PRE_PROCESSING, SUCCESS));
	
PRE_PROCESSING:
	IF (lastListChangeIndex <> currentListVersion) THEN
		cycleManager.proceedWith(ERROR);
		sort := CNM_ReturnTypes.SingleExecutionState.ERROR;
		RETURN;
	END_IF
	// Preprocess elements to create naturally sorted pairs
	preprocessResult := THIS^.preprocessElements(container, size);
	lastListChangeIndex := currentListVersion := currentListVersion + 1;
	IF preprocessResult = CNM_ReturnTypes.SingleExecutionResult.SUCCESS THEN
		// Pre-allocate buffer if container size changed
		
		// Allocate buffer for approximately n/2 elements (worst case)
		IF THIS^.mergeBuffer <> 0 THEN
			__DELETE(THIS^.mergeBuffer);
		END_IF
		THIS^.mergeBuffer := __NEW(__XWORD, SHR(size + 1, 1));
		cycleManager.assert.pointers.isNotNull(THIS^.mergeBuffer, message := 'arraylist twinsort: buffer allocation failed');
		// Preprocessing complete, start merging
		cycleManager.proceed();
	ELSIF preprocessResult = CNM_ReturnTypes.SingleExecutionResult.ABORTED THEN
		// Entire array was reversed (fully sorted)
		__DELETE(THIS^.mergeBuffer);
		cycleManager.proceedWith(SUCCESS);
	ELSE
		cycleManager.proceedWith(CNM_ReturnTypes.DefaultSteps.STEP.ERROR);
	END_IF		
MERGING:
	// Merge adjacent sequences of current width
	IF (lastListChangeIndex <> currentListVersion) THEN
		cycleManager.proceedWith(ERROR);
		sort := CNM_ReturnTypes.SingleExecutionState.ERROR;
		RETURN;
	END_IF
	THIS^.merge( container, size, mergeWidth);
	mergeWidth := SHL(mergeWidth, 1);
	lastListChangeIndex := currentListVersion := currentListVersion + 1;
	IF (mergeWidth >= size) THEN	
		// Sorting complete
		cycleManager.proceedWith(SUCCESS);
		__DELETE(THIS^.mergeBuffer);
	END_IF	
END_CASE

sort := cycleManager.state;
END_METHOD

END_FUNCTION_BLOCK

// ---- Lists/LinkedList/classes/LinkedListIterator/classes/InverseLinkedListIterator.TcPOU
{attribute 'enable_dynamic_creation'}
FUNCTION_BLOCK InverseLinkedListIterator EXTENDS AbstractLinkedListIterator
VAR	
	lastChangeVersion :__XWORD;
	lastExecute :BOOL;
END_VAR

PROPERTY className :CNM_AbstractObject.ClassName
GET
className := 'InverseLinkedListIterator';
END_GET
END_PROPERTY

(*

## Short summary

The constructor ``FB_init`` is needed to create an unique hash code.
The hash code is a pseudo random number create with a [xorshift](https://en.wikipedia.org/wiki/Xorshift) algorithm.
It can be overwritten on derivations, because it will be called implicit, ``SUPER^.FB_init()`` is not required.
For more information check: [Behavoir with derived function blocks](https://infosys.beckhoff.com/content/1033/tc3_plc_intro/5482088715.html?id=6983869892358031022).

.. <legal notes>

legal notes
=================
| SPDX-FileCopyrightText: © 2022 ekvip automation GmbH <info@ekvip.de>
| SPDX-License-Identifier: Apache-2.0
| For details check: Apache-2.0_

.. _Apache-2.0: https://www.apache.org/licenses/LICENSE-2.0

.. </legal notes>



*)
METHOD FB_init : BOOL
VAR_INPUT
	(* if TRUE, the retain variables are initialized (warm start / cold start)*)
	bInitRetains	: BOOL;
	(* if TRUE, the instance afterwards gets moved into the copy code (online change) *)
	bInCopyCode	: BOOL;
	(* list that is used to iterate*)
	list :REFERENCE TO LinkedList;
END_VAR
THIS^.direction := IterationDirection.BACKWARD;
END_METHOD

END_FUNCTION_BLOCK

// ---- Project Information/F_GetCompany.TcPOU
// This function has been automatically generated from the project information.
{attribute 'signature_flag' := '1073741824'}
{attribute 'TcGenerated'}
{attribute 'no-analysis'}
FUNCTION F_GetCompany : WSTRING
VAR_INPUT
	
END_VAR

F_GetCompany := "ekvip automation GmbH";

END_FUNCTION

// ---- Project Information/F_GetTitle.TcPOU
// This function has been automatically generated from the project information.
{attribute 'signature_flag' := '1073741824'}
{attribute 'TcGenerated'}
{attribute 'no-analysis'}
FUNCTION F_GetTitle : WSTRING
VAR_INPUT
	
END_VAR

F_GetTitle := "CNM_Collections";

END_FUNCTION

// ---- Project Information/F_GetVersion.TcPOU
// This function has been automatically generated from the project information.
{attribute 'signature_flag' := '1073741824'}
{attribute 'TcGenerated'}
{attribute 'no-analysis'}
FUNCTION F_GetVersion : ST_LibVersion
VAR_INPUT
	
END_VAR

F_GetVersion.iMajor := 0;
F_GetVersion.iMinor := 1;
F_GetVersion.iBuild := 1;
F_GetVersion.iRevision := 0;
F_GetVersion.sVersion := '0.1.1.0';
F_GetVersion.nFlags := 0;

END_FUNCTION
